RoboDK station: final.rdk

Station final. Poses are relative to the parent item; angles as X-Y-Z fixed-axis rotations.
